(* IEC 61131-3 sources: eCockpitGit/test_project/src/%F%00 Library/%F%Common Functions/%F%Math/%F%Difference, 12 files *)

(* ---- %POU%FU_bDiff.st ---- *)
//This function calculates the difference between two values, and outputs it positively
//
// +-----------+----------+----------+-----------------------------------------------------------------------------------------------------------------------+
// |**Version**|**Author**| **Date** |**Changes**                                                                                                            |
// +-----------+----------+----------+-----------------------------------------------------------------------------------------------------------------------+
// | 1         | NSN      | 02-08-18 | Creation                                                                                                              |
// +-----------+----------+----------+-----------------------------------------------------------------------------------------------------------------------+
FUNCTION FU_bDiff : BYTE
VAR_INPUT
	A			:BYTE;
	B			:BYTE;
END_VAR
(*%!%__DELIMITER__%!%*)
IF A > B THEN
	FU_bDiff			:=		A - B;
ELSE
	FU_bDiff			:=		B - A;
END_IF

(* ---- %POU%FU_diDiff.st ---- *)
//This function calculates the difference between two values, and outputs it positively
//
// +-----------+----------+----------+-----------------------------------------------------------------------------------------------------------------------+
// |**Version**|**Author**| **Date** |**Changes**                                                                                                            |
// +-----------+----------+----------+-----------------------------------------------------------------------------------------------------------------------+
// | 1         | NSN      | 02-08-18 | Creation                                                                                                              |
// +-----------+----------+----------+-----------------------------------------------------------------------------------------------------------------------+
FUNCTION FU_diDiff : DINT
VAR_INPUT
	A			:DINT;
	B			:DINT;
END_VAR
(*%!%__DELIMITER__%!%*)
IF A > B THEN
	FU_diDiff			:=		A - B;
ELSE
	FU_diDiff			:=		B - A;
END_IF

(* ---- %POU%FU_dwDiff.st ---- *)
//This function calculates the difference between two values, and outputs it positively
//
// +-----------+----------+----------+-----------------------------------------------------------------------------------------------------------------------+
// |**Version**|**Author**| **Date** |**Changes**                                                                                                            |
// +-----------+----------+----------+-----------------------------------------------------------------------------------------------------------------------+
// | 1         | NSN      | 02-08-18 | Creation                                                                                                              |
// +-----------+----------+----------+-----------------------------------------------------------------------------------------------------------------------+
FUNCTION FU_dwDiff : DWORD
VAR_INPUT
	A			:DWORD;
	B			:DWORD;
END_VAR

(*%!%__DELIMITER__%!%*)
IF A > B THEN
	FU_dwDiff			:=		A - B;
ELSE
	FU_dwDiff			:=		B - A;
END_IF

(* ---- %POU%FU_iDiff.st ---- *)
//This function calculates the difference between two values, and outputs it positively
//
// +-----------+----------+----------+-----------------------------------------------------------------------------------------------------------------------+
// |**Version**|**Author**| **Date** |**Changes**                                                                                                            |
// +-----------+----------+----------+-----------------------------------------------------------------------------------------------------------------------+
// | 1         | NSN      | 10-08-17 | Creation                                                                                                              |
// +-----------+----------+----------+-----------------------------------------------------------------------------------------------------------------------+
// | 1.1       | NSN      | 13-06-18 | Updated names and types                                                                                               |
// +-----------+----------+----------+-----------------------------------------------------------------------------------------------------------------------+
FUNCTION FU_iDiff : INT
VAR_INPUT
	A			:INT;
	B			:INT;
END_VAR

(*%!%__DELIMITER__%!%*)
IF A > B THEN
	FU_iDiff			:=		A - B;
ELSE
	FU_iDiff			:=		B - A;
END_IF

(* ---- %POU%FU_liDiff.st ---- *)
//This function calculates the difference between two values, and outputs it positively
//
// +-----------+----------+----------+-----------------------------------------------------------------------------------------------------------------------+
// |**Version**|**Author**| **Date** |**Changes**                                                                                                            |
// +-----------+----------+----------+-----------------------------------------------------------------------------------------------------------------------+
// | 1         | NSN      | 02-08-18 | Creation                                                                                                              |
// +-----------+----------+----------+-----------------------------------------------------------------------------------------------------------------------+
FUNCTION FU_liDiff : LINT
VAR_INPUT
	A			:LINT;
	B			:LINT;
END_VAR

(*%!%__DELIMITER__%!%*)
IF A > B THEN
	FU_liDiff			:=		A - B;
ELSE
	FU_liDiff			:=		B - A;
END_IF

(* ---- %POU%FU_lwDiff.st ---- *)
//This function calculates the difference between two values, and outputs it positively
//
// +-----------+----------+----------+-----------------------------------------------------------------------------------------------------------------------+
// |**Version**|**Author**| **Date** |**Changes**                                                                                                            |
// +-----------+----------+----------+-----------------------------------------------------------------------------------------------------------------------+
// | 1         | NSN      | 02-08-18 | Creation                                                                                                              |
// +-----------+----------+----------+-----------------------------------------------------------------------------------------------------------------------+
FUNCTION FU_lwDiff : LWORD
VAR_INPUT
	A			:LWORD;
	B			:LWORD;
END_VAR

(*%!%__DELIMITER__%!%*)
IF A > B THEN
	FU_lwDiff			:=		A - B;
ELSE
	FU_lwDiff			:=		B - A;
END_IF

(* ---- %POU%FU_siDiff.st ---- *)
//This function calculates the difference between two values, and outputs it positively
//
// +-----------+----------+----------+-----------------------------------------------------------------------------------------------------------------------+
// |**Version**|**Author**| **Date** |**Changes**                                                                                                            |
// +-----------+----------+----------+-----------------------------------------------------------------------------------------------------------------------+
// | 1         | NSN      | 02-08-18 | Creation                                                                                                              |
// +-----------+----------+----------+-----------------------------------------------------------------------------------------------------------------------+
FUNCTION FU_siDiff : SINT
VAR_INPUT
	A			:SINT;
	B			:SINT;
END_VAR

(*%!%__DELIMITER__%!%*)
IF A > B THEN
	FU_siDiff			:=		A - B;
ELSE
	FU_siDiff			:=		B - A;
END_IF

(* ---- %POU%FU_udiDiff.st ---- *)
//This function calculates the difference between two values, and outputs it positively
//
// +-----------+----------+----------+-----------------------------------------------------------------------------------------------------------------------+
// |**Version**|**Author**| **Date** |**Changes**                                                                                                            |
// +-----------+----------+----------+-----------------------------------------------------------------------------------------------------------------------+
// | 1         | NSN      | 02-08-18 | Creation                                                                                                              |
// +-----------+----------+----------+-----------------------------------------------------------------------------------------------------------------------+
FUNCTION FU_udiDiff : UDINT
VAR_INPUT
	A			:UDINT;
	B			:UDINT;
END_VAR

(*%!%__DELIMITER__%!%*)
IF A > B THEN
	FU_udiDiff			:=		A - B;
ELSE
	FU_udiDiff			:=		B - A;
END_IF

(* ---- %POU%FU_uiDiff.st ---- *)
//This function calculates the difference between two values, and outputs it positively
//
// +-----------+----------+----------+-----------------------------------------------------------------------------------------------------------------------+
// |**Version**|**Author**| **Date** |**Changes**                                                                                                            |
// +-----------+----------+----------+-----------------------------------------------------------------------------------------------------------------------+
// | 1         | NSN      | 02-08-18 | Creation                                                                                                              |
// +-----------+----------+----------+-----------------------------------------------------------------------------------------------------------------------+
FUNCTION FU_uiDiff : UINT
VAR_INPUT
	A			:UINT;
	B			:UINT;
END_VAR

(*%!%__DELIMITER__%!%*)
IF A > B THEN
	FU_uiDiff			:=		A - B;
ELSE
	FU_uiDiff			:=		B - A;
END_IF

(* ---- %POU%FU_uliDiff.st ---- *)
//This function calculates the difference between two values, and outputs it positively
//
// +-----------+----------+----------+-----------------------------------------------------------------------------------------------------------------------+
// |**Version**|**Author**| **Date** |**Changes**                                                                                                            |
// +-----------+----------+----------+-----------------------------------------------------------------------------------------------------------------------+
// | 1         | NSN      | 02-08-18 | Creation                                                                                                              |
// +-----------+----------+----------+-----------------------------------------------------------------------------------------------------------------------+
FUNCTION FU_uliDiff : ULINT
VAR_INPUT
	A			:ULINT;
	B			:ULINT;
END_VAR

(*%!%__DELIMITER__%!%*)
IF A > B THEN
	FU_uliDiff			:=		A - B;
ELSE
	FU_uliDiff			:=		B - A;
END_IF

(* ---- %POU%FU_usiDiff.st ---- *)
//This function calculates the difference between two values, and outputs it positively
//
// +-----------+----------+----------+-----------------------------------------------------------------------------------------------------------------------+
// |**Version**|**Author**| **Date** |**Changes**                                                                                                            |
// +-----------+----------+----------+-----------------------------------------------------------------------------------------------------------------------+
// | 1         | NSN      | 02-08-18 | Creation                                                                                                              |
// +-----------+----------+----------+-----------------------------------------------------------------------------------------------------------------------+
FUNCTION FU_usiDiff : USINT
VAR_INPUT
	A		:USINT;
	B		:USINT;
END_VAR

(*%!%__DELIMITER__%!%*)
IF A > B THEN
	FU_usiDiff			:=		A - B;
ELSE
	FU_usiDiff			:=		B - A;
END_IF

(* ---- %POU%FU_wDiff.st ---- *)
//This function calculates the difference between two values, and outputs it positively
//
// +-----------+----------+----------+-----------------------------------------------------------------------------------------------------------------------+
// |**Version**|**Author**| **Date** |**Changes**                                                                                                            |
// +-----------+----------+----------+-----------------------------------------------------------------------------------------------------------------------+
// | 1         | NSN      | 02-08-18 | Creation                                                                                                              |
// +-----------+----------+----------+-----------------------------------------------------------------------------------------------------------------------+
FUNCTION FU_wDiff : WORD
VAR_INPUT
	A			:WORD;
	B			:WORD;
END_VAR

(*%!%__DELIMITER__%!%*)
IF A > B THEN
	FU_wDiff			:=		A - B;
ELSE
	FU_wDiff			:=		B - A;
END_IF
